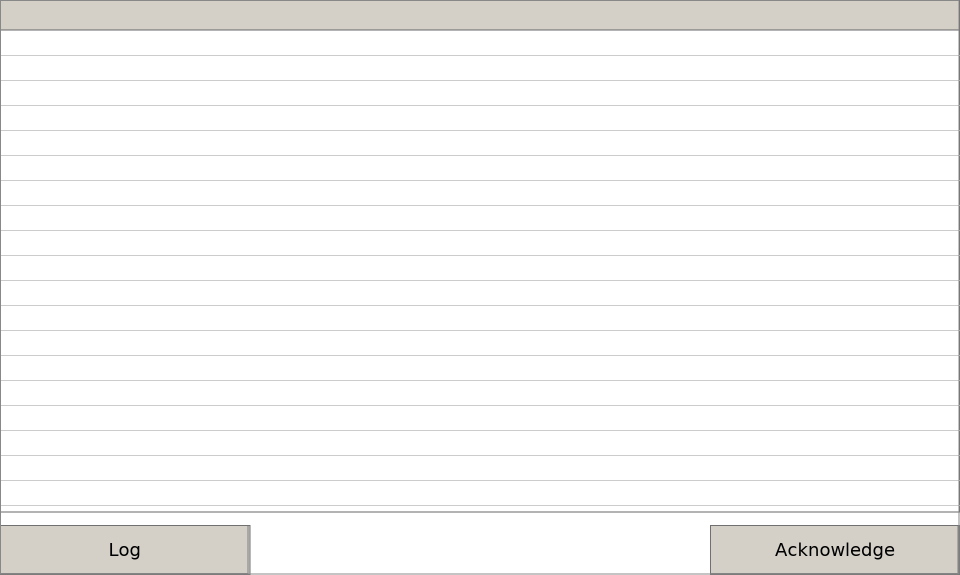
VISUALIZATION LogView  // 960x575
VAR_IN_OUT
	// NOTE: LogView table rows should match IBF_Utilities library parameter PAR_Utilities.MAX_FAULTS_IN_LOG
	fbLogView : FB_LogView;
	fbLogToDisk : FB_LogToDisk;
END_VAR
VAR
	bToggleLog : BOOL;
END_VAR
    TextEditor (0,0 960x512)
        p4127561890: Courier New
        p3844697057: fbLogToDisk.sCurrentLogFile
        p2773717400: Sys_Variables.Pulse1Sec
    Table (0,0 960x512), invisible if: bToggleLog, data array: fbLogView.arLog
        p3854506369: fbLogView.arLog[INDEX].sID
        p1892666644: fbLogView.arLog [INDEX].sDescription
        p338671338: fbLogView.arLog [INDEX].sStartTime
        p2170511999: fbLogView.arLog [INDEX].sEndTime
        p3723444502: fbLogView.arLog [INDEX].dColor_Bg
        p2685023577: fbLogView.arLog [INDEX].sID
        Columns.Column.[3].Template: fbLogView.arLog[INDEX].dColor_Bg
        Columns.Column.[2].Template: fbLogView.arLog[INDEX].dColor_Bg
        Columns.Column.[1].Template: fbLogView.arLog[INDEX].dColor_Bg
        Columns.Column.[0].Template: fbLogView.arLog[INDEX].dColor_Bg
    Button (710,525 250x50), "Acknowledge"
        tap fbLogView.bAcknowledge
    Button (0,525 250x50), "Log", pressed state: bToggleLog
        toggle bToggleLog
END_VISUALIZATION

(* stored: Version 1.1.0.1, ProductVersion 3.1.4024.11
   Visu LogView: Id {07ec0c4a-ff40-487e-8918-11af5123365d} *)
